END_CASE

IF i8Step > 0 AND i8Step < 80 THEN
	iStep																:= i8Step;
	Current_Step														:= iStep;
	sReactorError														:= SEL(product_line_temp_error, sReactorError, gsProductLineTempSensorError);
	sUtilityError														:= SEL(P_U01.steam_flow_error, sUtilityError, gsSteamFlowSensorError);
	A_Check_Process();
	i8Step																:= iStep;
END_IF
END_ACTION

ACTION A8_Bypass_1:
CASE i8Step OF	

	0:	;
		
	1:
		rTime1															:= _VALVE_TIME;
		i8Step															:= i8Step + 1;
		
	2:
		bTimer1															:= TRUE;
		IF tonTimer1.Q THEN
			bTimer1														:= FALSE;
			i8Step														:= 99;
		END_IF
	
	99:
		bBypassDone														:= TRUE;											// 5
		Current_Step													:= 0;
		i8Step															:= 0;
	
END_CASE

IF i8Step > 0 AND i8Step < 80 THEN
	iStep																:= i8Step;
	Current_Step														:= iStep;
	A_Check_Process();
	i8Step																:= iStep;
END_IF
END_ACTION

END_FUNCTION_BLOCK

(* stored: Version 1.1.0.1, ProductVersion 3.1.4024.12
   POU FB_Reactor_Set: Id {7a14df60-c425-4007-b6c2-e2f870fc0897}, SpecialFunc None
   Action A_Check_Process: Id {6ec7fe9a-742c-414a-a60e-a55eaa5d8982}
   Action A_Clear_Variables: Id {0dbcb2f7-e4a4-40b8-8807-7ed3a1095350}
   Action A_Drain_Reactor_Set: Id {1d4eeb92-89ea-4631-b611-8a78ca35984b}
   Action A_Idle: Id {f9da58c1-f853-41c1-a061-a5899835c823}
   Action A_Reactor_Set_IO: Id {25429ff6-89a6-49d1-95df-80da2347faf4}
   Action A_Reset: Id {f03b698c-165a-4253-9d0f-30912c71aaa9}
   Action A2_DoorCycle_1: Id {7c2960b8-c74b-4c37-9302-9cbfbf90678e}
   Action A2_DoorCycle_OLD: Id {3eff279f-9b41-4145-b6ae-283999c67d9f}
   Action A3_PositivePressure_1: Id {12952df9-63c1-4f1a-9695-efe190e64781}
   Action A3_PositivePressure_OLD: Id {cd930d60-1df9-4a9e-a703-94a83a9f89d2}
   Action A4_Repressurization: Id {fb715d4f-ecdc-4079-89b7-548849d9330a}
   Action A4_Repressurization_1: Id {026d52b5-f57f-48eb-ad87-a9da6d8e7d67}
   Action A4_Repressurization_OLD: Id {754a3da5-03af-4044-b9fa-b4481f24ea64}
   Action A5_Adsorption: Id {eff2fd60-8c5e-4677-a3e6-5e563647498b}
   Action A5_Adsorption_1: Id {4becb6ac-c555-4f6d-8c9b-3eaf6fcd7a35}
   Action A5_Adsorption_OLD: Id {b320dbf0-895a-4407-bdf8-77442686e4f4}
   Action A6_Evacuation: Id {435cb2e1-0f88-42fa-90cb-927b82ea0edf}
   Action A6_Evacuation_1: Id {1f183e1d-b96d-4bce-9f37-a84d41018cf9}
   Action A6_Evacuation_OLD: Id {f61283cf-bd53-411a-b295-99a0bade7a7d}
   Action A7_Desorption: Id {e1929abd-aa53-4940-b6ab-ecb493f839a5}
   Action A7_Desorption_1: Id {33223d60-8bc5-49dd-a111-128ac5fbf786}
   Action A7_Desorption_OLD: Id {64b66c6d-be92-49a7-80c1-a34cbffc87f4}
   Action A8_Bypass: Id {79bb11fb-ab2e-48df-8558-afb0d41e5d1b}
   Action A8_Bypass_1: Id {d961da16-3975-47b6-8535-b84ca3745368} *)
